TYPE ST_HW_InputsSickScanner_CLV690 :
STRUCT
	DeviceReady		: BOOL;
	GoodRead		: BOOL;
	NoRead			: BOOL;
	ConfMessageIn	: ARRAY[0..31] OF BYTE; // Message
END_STRUCT
END_TYPE

(* stored: Version 1.1.0.1, ProductVersion 3.1.4024.4
   DUT ST_HW_InputsSickScanner_CLV690: Id {e846b8ca-d825-41e5-a249-06e5f1e6e7da} *)
